(* PLC project IntralogisticsLab, Intralogistics Learning Lab CODESYS V3.5 SP19 3.5.19.0 *)
(* stored: creationDateTime 2025-08-25T12:00:00, modificationDateTime 2025-08-25T12:00:00 *)

TYPE DUT_SystemState : (SYSTEM_STOPPED := 0, SYSTEM_STARTING := 1, SYSTEM_RUNNING := 2, SYSTEM_STOPPING := 3, SYSTEM_ERROR := 4, SYSTEM_MANUAL := 5);
END_TYPE

TYPE DUT_RobotState : (ROBOT_IDLE := 0, ROBOT_MOVING_TO_BIN := 1, ROBOT_AT_BIN := 2, ROBOT_PICKING := 3, ROBOT_MOVING_TO_STATION := 4, ROBOT_AT_STATION := 5, ROBOT_PLACING := 6, ROBOT_RETURNING_HOME := 7, ROBOT_ERROR := 8);
END_TYPE

TYPE DUT_ConveyorStatus : (CONVEYOR_STOPPED := 0, CONVEYOR_RUNNING := 1, CONVEYOR_FAULT := 2, CONVEYOR_MAINTENANCE := 3);
END_TYPE

TYPE DUT_RFIDStatus : (RFID_IDLE := 0, RFID_READING := 1, RFID_VALID_READ := 2, RFID_ERROR := 3, RFID_NO_TAG := 4);
END_TYPE

TYPE DUT_StationType : (STATION_NONE := 0, STATION_RECEIVING := 1, STATION_ASSEMBLY := 2, STATION_WAREHOUSE := 3);
END_TYPE

TYPE DUT_ConveyorData : STRUCT
  Status : ?;
  Motor_Command : ?;
  Speed_Setpoint : ?;
  Entry_Sensor : ?;
  Exit_Sensor : ?;
  Run_Timer : ?;
  Fault_Code : ?;
  Item_Count : ?;
  Auto_Mode : ?;
END_STRUCT;
END_TYPE

TYPE DUT_RobotData : STRUCT
  Current_State : ?;
  Target_Bin : ?;
  Target_Station : ?;
  Position_X : ?;
  Position_Y : ?;
  Position_Z : ?;
  At_Home : ?;
  At_Target : ?;
  Gripper_Open : ?;
  Gripper_Closed : ?;
  Moving : ?;
  Error_Code : ?;
  Operation_Timer : ?;
  Enable_Command : ?;
  Reset_Command : ?;
END_STRUCT;
END_TYPE

TYPE DUT_RFIDData : STRUCT
  Status : ?;
  Tag_Present : ?;
  Tag_ID : ?;
  Read_Command : ?;
  Enable_Command : ?;
  Ready : ?;
  Read_Timer : ?;
  Error_Code : ?;
  Valid_Read_Count : ?;
  Error_Count : ?;
END_STRUCT;
END_TYPE

PROGRAM MAIN
  VAR
    System_Initialize : ?;
    System_Enable : ?;
    System_Reset : ?;
    Manual_Mode_Request : ?;
    FB_Safety : ?;
    FB_Conveyors : ?;
    FB_Robot : ?;
    FB_PickControl : ?;
    FB_RFID : ?;
    FB_Beacons : ?;
    Robot_Data : ?;
    System_Ready : ?;
    All_Systems_OK : ?;
    Any_System_Error : ?;
    Cycle_Counter : ?;
    Uptime_Counter : ?;
    Heartbeat_Counter : ?;
    HMI_System_Start : ?;
    HMI_System_Stop : ?;
    HMI_System_Reset : ?;
    HMI_Manual_Mode : ?;
    Init_Timer : ?;
    Init_Complete : ?;
  END_VAR

            
              
            
          
END_PROGRAM

FUNCTION_BLOCK FB_SafetySystem
  VAR_INPUT
    System_Enable : ?;
    Manual_Reset : ?;
    Bypass_Mode : ?;
  END_VAR
  VAR_OUTPUT
    Safety_OK : ?;
    Emergency_Stop : ?;
    Reset_Required : ?;
    System_Safe : ?;
    Fault_Code : ?;
  END_VAR

END_FUNCTION_BLOCK

CONFIGURATION Config0
  RESOURCE Res0 ON PLC
    TASK Main(INTERVAL := T#100ms, PRIORITY := 0);
    PROGRAM Inst0 : MAIN;
  END_RESOURCE
END_CONFIGURATION
